TYPE StateTimeStamp :
STRUCT
	Station: DINT;
	ID: DINT;
	State: DINT;
	TimeLo: UDINT;
	TimeHi: UDINT;
END_STRUCT
END_TYPE

(* stored: Version 1.1.0.1, ProductVersion 3.1.4024.9
   DUT StateTimeStamp: Id {37043554-7926-468f-9b0e-2a2649e50372} *)
